TYPE
    UNI_CylinderList :
    UNION
        arCylinder : ARRAY[1..udiMax_CylinderNum] OF FB_Cylinder;
        List       : ST_CylinderList;
    END_UNION
END_TYPE

(* stored: Version 1.1.0.1, ProductVersion 3.1.4024.13
   DUT UNI_CylinderList: Id {2d6f0041-738f-43a4-8e43-0d3aecc2acb3} *)
